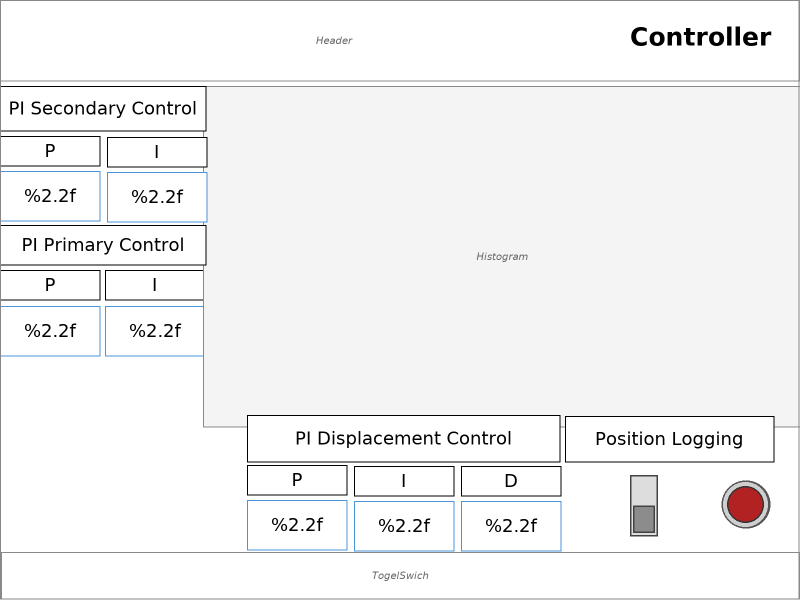
VISUALIZATION Screen_PID_Control  // 800x600
    Rectangle (0,306 100x50), "%2.2f", text variable: HMI.bP_PI
        OnMouseDown: write HMI.bProtielGainP_DC via VisuDialogs.Numpad, min 0, max 40
    Frame (-132,0 932x81)
        shows Header()
    Rectangle (105,306 100x50), "%2.2f", text variable: HMI.bI_PI
        OnMouseDown: write HMI.bI_PI via VisuDialogs.Numpad, min 0, max 40
    Frame (1,552 799x47)
        shows TogelSwich()
    Rectangle (0,270 100x30), "P", text variable: HMI.bData1
    Rectangle (105,270 100x30), "I", text variable: HMI.bData1
    Histogram (203,86 599x341), scale format: %.1f, scale 1..2
        p1518820177: HMI.arrPayLoadPositions
        p102497268: HMI.arrPayLoadPositions
        p788070771: ARRAY [1..100] OF LREAL
    Textfield (623,20 156x33), "Controller"
    Rectangle (0,225 206x40), "PI Primary Control"
    Rectangle (247,415 313x47), "PI Displacement Control"
    Rectangle (0,86 206x45), "PI Secondary Control"
    Rectangle (0,171 100x50), "%2.2f", text variable: HMI.bProtielGainP_SC
        OnMouseDown: write HMI.bProtielGainP_SC via VisuDialogs.Numpad, min 0, max 100
    Rectangle (0,136 100x30), "P", text variable: HMI.bData1
    Rectangle (107,172 100x50), "%2.2f", text variable: HMI.bProtielGainI_SC
        OnMouseDown: write HMI.bProtielGainI_SC via VisuDialogs.Numpad, min 0, max 100
    Rectangle (107,137 100x30), "I", text variable: HMI.bData1
    Rectangle (247,500 100x50), "%2.2f", text variable: HMI.bProtielGainP_DC
        OnMouseDown: write HMI.bProtielGainP_DC via VisuDialogs.Numpad, min 0, max 100
    Rectangle (247,465 100x30), "P", text variable: HMI.bData1
    Rectangle (354,501 100x50), "%2.2f", text variable: HMI.bProtielGainI_DC
        OnMouseDown: write HMI.bProtielGainI_DC via VisuDialogs.Numpad, min 0, max 1200
    Rectangle (354,466 100x30), "I", text variable: HMI.bData1
    Rectangle (461,501 100x50), "%2.2f", text variable: HMI.bProtielGainD_DC
        OnMouseDown: write HMI.bProtielGainD_DC via VisuDialogs.Numpad, min 0, max 250
    Rectangle (461,466 100x30), "D", text variable: HMI.bData1
    DipSwitch (575,475 138x61), variable: HMI.bSwichForPlot, behaviour: TOGGLE, style: Switch-DipSwitch-Gray
    Rectangle (565,416 209x46), "Position Logging", text variable: HMI.bData1
    Lamp1 (719,477 55x55), variable: HMI.bSwichForPlot, invisible if: not HMI.bSwichForPlot, style: Lamp-Lamp1-Green
    Lamp1 (718,477 55x55), variable: not HMI.bSwichForPlot, invisible if: HMI.bSwichForPlot, style: Lamp-Lamp1-Red
END_VISUALIZATION

(* stored: Version 1.1.0.1, ProductVersion 3.1.4024.12
   Visu Screen_PID_Control: Id {caff239a-c461-4107-bcc6-2cd12493fdac} *)
